% RSLogix 500 project Q12.RSS, saved by version 8.30.00.16 %
PROJECT "Q12"    % processor: Bul.1763 MicroLogix 1100 Series B %

PROGRAM FILES
  LAD 2   6 rungs

DATA FILES
  O0 OUTPUT  4 elements
  I1 INPUT  6 elements
  S2 STATUS  66 elements
  B3 BINARY  1 elements
  T4 TIMER  1 elements
  C5 COUNTER  1 elements
  R6 CONTROL  1 elements
  N7 INTEGER  1 elements
  F8 FLOAT  1 elements

LADDER 2
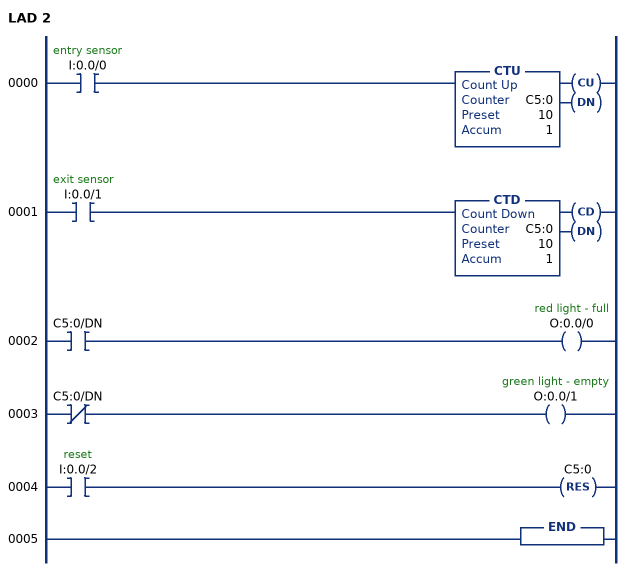
% Rung: 0 %
SOR XIC I:0.0/0 CTU C5:0 10 1 EOR
%   I:0.0/0  "entry sensor" %
% Rung: 1 %
SOR XIC I:0.0/1 CTD C5:0 10 1 EOR
%   I:0.0/1  "exit sensor" %
% Rung: 2 %
SOR XIC C5:0/DN OTE O:0.0/0 EOR
%   O:0.0/0  "red light - full" %
% Rung: 3 %
SOR XIO C5:0/DN OTE O:0.0/1 EOR
%   O:0.0/1  "green light - empty" %
% Rung: 4 %
SOR XIC I:0.0/2 RES C5:0 EOR
%   I:0.0/2  "reset" %
% Rung: 5 %
SOR END EOR

DATA TABLE (non-zero values as saved)
DATA C5
% .PRE .ACC %
% C5:0 % 10 1
